FUNCTION_BLOCK FB_SimulatedDigOutOpen_AFO IMPLEMENTS ITF_Schuif_DigOutOpen_AFO
VAR
	internalState : BOOL := FALSE;
END_VAR

METHOD set : BOOL
VAR_INPUT
	state : BOOL;
END_VAR
internalState := state;
END_METHOD

END_FUNCTION_BLOCK

(* stored: Version 1.1.0.1, ProductVersion 3.1.4026.8
   POU FB_SimulatedDigOutOpen_AFO: Id {344ce2d3-5a32-466b-a26c-1b17147eb765}, SpecialFunc None
   Method set: Id {4c281178-76bf-4d71-87b0-d914c8aff672} *)
